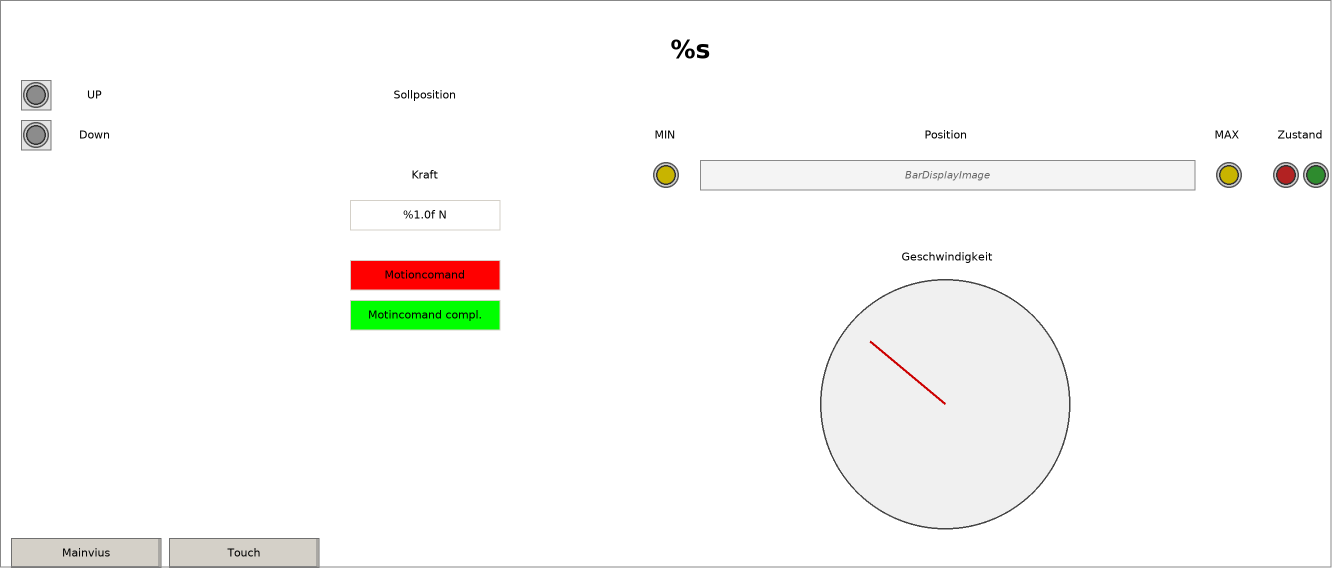
VISUALIZATION Visu_Achse  // 1332x568
VAR_IN_OUT
	Axis :FBCylTronicCylinder;
END_VAR
    Label (700,120 495x30), "Position"
    PushSwitch (20,80 32x30), variable: Axis.bUP, invisible if: NOT Axis.bManual or GVL.Achsenkontrolle, behaviour: TAP, style: Switch-PushSwitch-Gray
    PushSwitch (20,120 32x30), variable: Axis.bDOWN, invisible if: NOT Axis.bManual or GVL.Achsenkontrolle, behaviour: TAP, style: Switch-PushSwitch-Gray
    Label (60,80 69x30), "UP", invisible if: NOT Axis.bManual or GVL.Achsenkontrolle
    Label (60,120 69x30), "Down", invisible if: NOT Axis.bManual or GVL.Achsenkontrolle
    Label (350,80 150x30), "Sollposition"
    BarDisplayImage (700,160 495x30), value: Axis.ActualPosition, style: BarDisplayImage-Gray, scale format: %.0f, scale 0..200
    Lamp1 (1270,160 32x30), variable: Axis.WarningActive, style: Lamp-Lamp1-Red
    Lamp1 (1300,160 32x30), variable: Axis.Ready, style: Lamp-Lamp1-Green
    Label (350,160 150x30), "Kraft"
    Textfield (350,200 150x30), "%1.0f N", text variable: Axis.ActualForce
    Label (872,242 150x30), "Geschwindigkeit"
    Meter360 (820,279 250x250), value: Axis.ActualSpeed, style: Meter-Meter360-Gray, scale format: %.0f, scale -220..220
    Lamp1 (650,160 32x30), variable: Axis.LimitSwitchIn, style: Lamp-Lamp1-Yellow
    Lamp1 (1213,160 32x30), variable: Axis.LimitSwitchOut, style: Lamp-Lamp1-Yellow
    Textfield (350,300 150x30), "Motincomand compl.", invisible if: NOT Axis.MotionCommandCompleted
    Textfield (350,260 150x30), "Motioncomand", invisible if: NOT Axis.MotionModeActive
    Label (635,120 60x30), "MIN"
    Label (1197,120 60x30), "MAX"
    Label (1270,120 60x30), "Zustand"
    Button (11,538 150x30), "Mainvius"
        OnMouseDown: change screen: Mainvisu
    Button (169,538 150x30), "Touch"
        OnMouseDown: change screen: FigurePlayer
    Textfield (297,12 787x74), "%s", text variable: Axis.stAxisName
END_VISUALIZATION

(* stored: Version 1.1.0.1, ProductVersion 3.1.4024.12
   Visu Visu_Achse: Id {36645ab4-a1e8-4b07-807e-2f552a651f05} *)
